Universal Robots URScript: vino 4binf.script

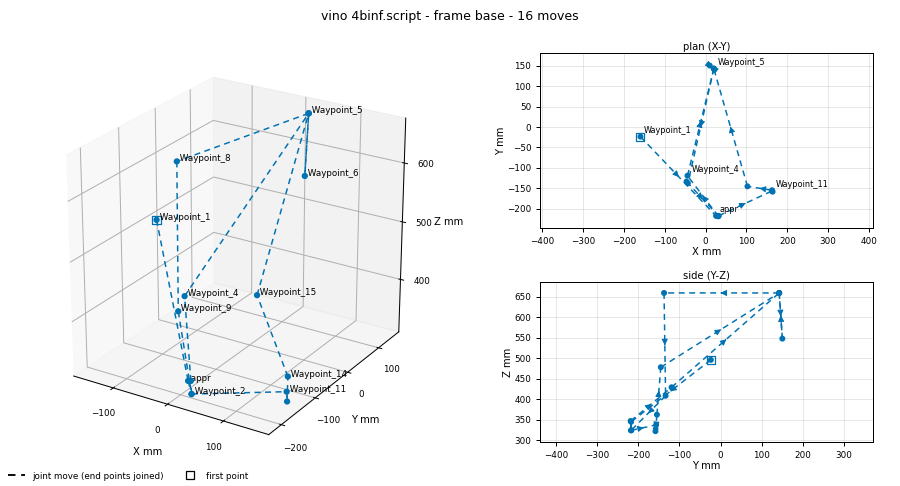
[picture p0: tool path of vino 4binf.script in frame base, 16 of 17 moves have a stored position in this frame; points joined in program order, loops and branches not executed]
def vino_4binf():
  set_gravity([0.0, 0.0, 9.82])
  set_safety_mode_transition_hardness(1)
  step_count_7828767f_f0a1_4da8_ad6d_1d539f3a6eb4 = 0.0
  thread Step_Counter_Thread_a07dad3b_d2d5_4c2a_9756_74ff32e0ed35():
    while (True):
      step_count_7828767f_f0a1_4da8_ad6d_1d539f3a6eb4 = step_count_7828767f_f0a1_4da8_ad6d_1d539f3a6eb4 + 1.0
      sync()
    end
  end
  run Step_Counter_Thread_a07dad3b_d2d5_4c2a_9756_74ff32e0ed35()
  set_tcp(p[0.0,0.0,0.155,0.0,0.0,0.0])
  set_payload(1.1, [0.0, 0.0, 0.06])
  set_standard_analog_input_domain(0, 1)
  set_standard_analog_input_domain(1, 1)
  set_tool_analog_input_domain(0, 1)
  set_tool_analog_input_domain(1, 1)
  set_analog_outputdomain(0, 0)
  set_analog_outputdomain(1, 0)
  set_input_actions_to_default()
  set_tool_voltage(24)
  global Plane_obliquo=p[0.09998422840375992,0.0999895685224925,0.14997740118490663,-0.1474295993751028,-0.061308860415087624,0.7833703634583852]
  global Plane_orizz=p[9.515322773469715E-6,0.2500097097193357,0.14997678393289224,-8.204102312405902E-5,-5.45201065398691E-5,1.2537983658861858E-5]
  global Plane_vert=p[2.5528049992290395E-5,0.45000115403946234,0.014993315552056186,1.5707062492170034,-1.3296462557657132E-4,1.823233379452444E-4]
  # begin: URCap Installation Node
  #   Source: OnRobot, 6.0.3, OnRobot A/S
  #   Type: OnRobot Setup
  sleep(1)
  if (False):
    global sg_Busy = 0
    global sg_Depth = 0
    global sg_Width = 0
  end
  ON_CONN_SHIFT_BOOL = 64
  ON_CONN_SHIFT_INT = 24
  ON_CONN_SHIFT_FLOAT = 24
  ON_CONN_REG_SUM_BOOL = 2
  ON_CONN_REG_SUM_INT = 4
  ON_CONN_REG_SUM_FLOAT = 3
  ON_TOOL_SHIFT_BOOL = 64
  ON_TOOL_SHIFT_INT = 25
  ON_TOOL_SHIFT_FLOAT = 24
  ON_TOOL_SHIFT_BOOL_ARR = [64, 66, 66]
  ON_TOOL_SHIFT_INT_ARR = [25, 28, 28]
  ON_TOOL_SHIFT_FLOAT_ARR = [24, 27, 27]
  ON_TOOL_REG_SUM_BOOL = 2
  ON_TOOL_REG_SUM_INT = 3
  ON_TOOL_REG_SUM_FLOAT = 3
  ON_REGISTERS_SPEEDL_FLOAT = 0
  ON_REG_USE_TOOL = False
  ON_DI_SINGLE = 0
  ON_DI_PRIMARY = 1
  ON_DI_SECONDARY = 2
  ON_DI_DUAL = 3
  on_robot_type = 3
  on_robot_cycle = 8.0
  on_conn_ip = "localhost"
  on_tool_ip = "localhost"
  on_device_socket_port = 51234
  on_conn_xmlrpc = rpc_factory("xmlrpc", "http://localhost:41414")
  on_tool_xmlrpc = rpc_factory("xmlrpc", "http://localhost:41414")
  on_RPC = rpc_factory("xmlrpc", "http://127.0.0.1:31416")
  ON_DEBUG_LOG = False
  on_isMetric = True
  on_toolConnector = True
  on_ioqc = True
  on_dual = False
  on_computebox = False
  on_devices = 1
  on_gripper = [False, False, False]
  on_custom_tcp_id = "none"
  on_custom_tcp_enabled = False
  speedlTime = 0.001
  on_ft = False
  sg_index = 0
  on_gripper[sg_index] = True
  #======    OnRobot Globals    ======#

  ON_MATH_PI=3.141593
  ON_ZEROPOSE=p[0.0,0.0,0.0,0.0,0.0,0.0]
  ON_ZEROFRAME=p[0.0,0.0,0.0,0.0,0.0,0.0]
  ON_ZERO3D=[0.0,0.0,0.0]
  ON_ZERO6D=[0.0,0.0,0.0,0.0,0.0,0.0]
  ON_ZERO8D=[0.0,0.0,0.0,0.0,0.0,0.0,0.0,0.0]
  ON_FALSE3D=[False,False,False]
  ON_FALSE6D=[False,False,False,False,False,False]
  ON_FALSE8D=[False,False,False,False,False,False,False,False]
  global on_return=0
  on_speedL=ON_ZERO6D
  on_speedBase=ON_ZERO6D
  on_speedVect=ON_ZERO6D
  on_speedExtra=ON_ZERO6D
  on_speedCB=ON_ZERO6D
  on_speedGecko=ON_ZERO6D
  on_RTDE_error=0
  on_RTDE_tool_error=0
  on_dataProcess_thrd=0
  ON_DEVICE_ID_MISSING=0
  ON_INIT_WATCHDOG_HZ=5
  ON_INIT_TIMEOUT=2000
  on_robot_TCP_offset=ON_ZEROFRAME
  on_tcp_offset_actual=ON_ZEROFRAME
  on_cog_actual=ON_ZEROFRAME
  on_mass_actual=0.0
  on_robot_mount=[0.0,0.0]

  #======    End of OnRobot Globals    ======#
  #======    OnRobot SG Globals    ======#

  SG_DEVICE_ID=80
  sg_Width_arr=[0,0,0]
  sg_Depth_arr=[0,0,0]
  sg_DepthRel_arr=[0,0,0]
  sg_device_id_arr=[0,0,0]
  sg_product_code_arr=[0,0,0]
  sg_Status_arr=[0,0,0]
  sg_Busy_arr=[False,False,False]
  sg_Initialized_arr=[False,False,False]
  sg_Grip_command_arr=[False,False,False]
  sg_tool_id_arr=[0,0,0]

  sg_Width=0
  sg_Depth=0
  sg_Busy=False
  def get_sg_Width():
  return sg_Width
  end
  def get_sg_Depth():
  return sg_Depth
  end
  def get_sg_Busy():
  return sg_Busy
  end


  #======    End of OnRobot SG Globals    ======#
  #======    OnRobot Interface Messages    ======#

  on_devices_primary_log="OnRobot Devices"
  on_devices_secondary_log="OnRobot Secondary Device"
  on_program_halted="<br>Program halted."
  on_device_error_title="OnRobot - Device error"
  on_install_error="OnRobot Setup is not correct.<br>Check the status in the OnRobot Setup page in the Installation Tab.<br>Program halted."
  on_device_missing="No device connected.<br>Program halted."
  cb_device_missing="No OnRobot Compute Box connected.<br>Program halted."
  ft_device_missing="No OnRobot FT sensor or license detected.<br>Program halted."
  hex_device_missing="No HEX sensor connected.<br>Program halted."
  rg2ft_device_missing="No RG2-FT gripper connected.<br>Program halted."
  rg_device_missing="No RG gripper connected.<br>Program halted."
  vg_device_missing="No VG gripper connected.<br>Program halted."
  gg_device_missing="No Gecko Gripper connected.<br>Program halted."
  sg_device_missing="No Soft Gripper connected.<br>Program halted."
  tfg_device_missing="No 3FG gripper connected.<br>Program halted."
  sdr_device_missing="No OnRobot Sander connected.<br>Program halted."
  twofg_device_missing="No 2FG gripper connected.<br>Program halted."
  vgp_device_missing="No VGP gripper connected.<br>Program halted."
  mg_device_missing="No Magnetic Gripper connected.<br>Program halted."
  fgp_device_missing="No 2FGP20 Gripper connected.<br>Program halted."
  eyes_device_missing="No OnRobot Eyes connected.<br>Program halted."
  on_xmlrpc_start_ip="Connecting to OnRobot XML-RPC Server:"
  on_java_comm_error_textmsg_title="OnRobot - Communication error:"
  on_java_comm_controlsocket_open_error="Socket 'javaSocket' opening was unsuccessful."
  on_java_comm_error_title="OnRobot - Communication error"
  on_java_comm_socket_open_error="Establishing connection with the URCap was timed out.<br>Check the status in the OnRobot Setup page in the Installation Tab.<br>Program halted."
  on_rtde_feed_error_textmsg_title="OnRobot - RTDE error:"
  on_rtde_feed_error="RTDE feed error. OnRobot device count mismatch.<br>Program halted."
  on_rtde_feed_tool_error="Tool RTDE feed error. OnRobot device count mismatch.<br>Program halted."
  on_rtde_feed_open_error_textmsg="Socket 'rtdeFeed' opening was unsuccessful."
  on_rtde_feed_error_title="OnRobot - RTDE error"
  on_rtde_feed_count_error="Invalid RTDE offset setup detected. Please check RTDE Offsets at the OnRobot Setup page in the Installation Tab.<br>Program halted."
  on_rtde_feed_open_error="Establishing connection with the devices was timed out.<br>Ensure that the OnRobot devices are operational, and check the status in the OnRobot Setup page in the Installation Tab."

  #======    End of OnRobot Interface Messages    ======#
  #======    OnRobot Interface    ======#

  on_portopened_javaSocket=False
  on_rtde_feed_opened=False
  on_dataProcess_running=False
  def on_missing():
  popup(on_device_missing,title=on_device_error_title,error=True,blocking=False)
  halt
  end
  def cb_missing():
  popup(cb_device_missing,title=on_device_error_title,error=True,blocking=False)
  halt
  end
  def ft_missing():
  popup(ft_device_missing,title=on_device_error_title,error=True,blocking=False)
  halt
  end
  def hex_missing():
  popup(hex_device_missing,title=on_device_error_title,error=True,blocking=False)
  halt
  end
  def rg2ft_missing():
  popup(rg2ft_device_missing,title=on_device_error_title,error=True,blocking=False)
  halt
  end
  def rg_missing():
  popup(rg_device_missing,title=on_device_error_title,error=True,blocking=False)
  halt
  end
  def vg_missing():
  popup(vg_device_missing,title=on_device_error_title,error=True,blocking=False)
  halt
  end
  def gg_missing():
  popup(gg_device_missing,title=on_device_error_title,error=True,blocking=False)
  halt
  end
  def sg_missing():
  popup(sg_device_missing,title=on_device_error_title,error=True,blocking=False)
  halt
  end
  def tfg_missing():
  popup(tfg_device_missing,title=on_device_error_title,error=True,blocking=False)
  halt
  end
  def sdr_missing():
  popup(sdr_device_missing,title=on_device_error_title,error=True,blocking=False)
  halt
  end
  def twofg_missing():
  popup(twofg_device_missing,title=on_device_error_title,error=True,blocking=False)
  halt
  end
  def vgp_missing():
  popup(vgp_device_missing,title=on_device_error_title,error=True,blocking=False)
  halt
  end
  def mg_missing():
  popup(mg_device_missing,title=on_device_error_title,error=True,blocking=False)
  halt
  end
  def fgp_missing():
  popup(fgp_device_missing,title=on_device_error_title,error=True,blocking=False)
  halt
  end
  def eyes_missing():
  popup(eyes_device_missing,title=on_device_error_title,error=True,blocking=False)
  halt
  end
  def on_portclose_javaSocket():
  socket_close("javaSocket")
  on_portopened_javaSocket=False
  end
  def on_portopen_javaSocket():
  on_portclose_javaSocket()
  on_portopened_javaSocket=socket_open("127.0.0.1",44005,"javaSocket")
  if not on_portopened_javaSocket:
  textmsg(on_java_comm_error_textmsg_title,on_java_comm_controlsocket_open_error)
  popup(on_java_comm_socket_open_error,title=on_java_comm_error_title,error=True,blocking=False)
  halt
  end
  end
  on_conn_rtde_feed_name="rtdeFeedConn"
  on_tool_rtde_feed_name="rtdeFeedTool"
  def on_rtde_feed_close(rtdeFeedName):
  socket_close(rtdeFeedName)
  on_rtde_feed_opened=False
  end
  def on_rtde_feed_open(deviceIP,rtdeFeedName,regStart,regSum,regSpeedl):
  on_rtde_feed_close(rtdeFeedName)
  if((regStart[0]+regSum[0])>128)or((regStart[1]+regSum[1])>48)or((regStart[2]+regSum[2])>48):
  popup(on_rtde_feed_count_error,title=on_rtde_feed_error_title,error=True,blocking=False)
  textmsg(str_cat("RegStart: ",regStart),str_cat("  -  RegSum: ",regSum))
  halt
  end
  on_rtde_feed_opened=socket_open(deviceIP,on_device_socket_port,rtdeFeedName)
  if not on_rtde_feed_opened:
  on_rtde_feed_opened=socket_open(deviceIP,on_device_socket_port,rtdeFeedName)
  end
  if not on_rtde_feed_opened:
  textmsg(on_rtde_feed_error_textmsg_title,on_rtde_feed_open_error_textmsg)
  popup(on_rtde_feed_open_error,title=on_rtde_feed_error_title,error=True,blocking=False)
  halt
  end
  socket_send_int(regStart[0],rtdeFeedName)
  socket_send_int(regSum[0],rtdeFeedName)
  socket_send_int(regStart[1],rtdeFeedName)
  socket_send_int(regSum[1],rtdeFeedName)
  socket_send_int(regStart[2],rtdeFeedName)
  socket_send_int(regSum[2],rtdeFeedName)
  socket_send_int(regSpeedl,rtdeFeedName)
  socket_send_int(on_devices,rtdeFeedName)
  end
  def on_dataRead():
  enter_critical
  on_RTDE_error=read_input_integer_register(ON_CONN_SHIFT_INT)
  if(ON_REG_USE_TOOL):
  on_RTDE_tool_error=read_input_integer_register(ON_TOOL_SHIFT_INT_ARR[0])
  end
  exit_critical
  end
  def on_set_rtde_watchdog(updateHz=ON_INIT_WATCHDOG_HZ):
  local effect="stop"
  if(updateHz<1):
  effect="ignore"
  end
  watchdog_conn_reg_str=str_cat("input_int_register_",ON_CONN_SHIFT_INT)
  rtde_set_watchdog(watchdog_conn_reg_str,updateHz,effect)
  if(ON_REG_USE_TOOL):
  watchdog_tool_reg_str=str_cat("input_int_register_",ON_TOOL_SHIFT_INT_ARR[0])
  rtde_set_watchdog(watchdog_tool_reg_str,updateHz,effect)
  end
  if ON_DEBUG_LOG:
  local update_str=str_cat(" "+effect+" watchdog set to [Hz]: ",updateHz)
  textmsg(watchdog_conn_reg_str,update_str)
  if(ON_REG_USE_TOOL):
  local update_str=str_cat(" "+effect+" watchdog set to [Hz]: ",updateHz)
  textmsg(watchdog_tool_reg_str,update_str)
  end
  end
  end
  def on_speedCB_get():
  return[on_speedCB[0],on_speedCB[1],on_speedCB[2],on_speedCB[3],on_speedCB[4],on_speedCB[5]]
  end
  def on_speedGecko_get():
  local speedExtra=ON_ZERO6D
  if on_speedl_for_gecko:
  speedExtra=[on_speedGecko[0],on_speedGecko[1],on_speedGecko[2],on_speedGecko[3],on_speedGecko[4],on_speedGecko[5]]
  end
  return speedExtra
  end
  def on_speedGecko_set(speedGecko):
  on_speedGecko=[speedGecko[0],speedGecko[1],speedGecko[2],speedGecko[3],speedGecko[4],speedGecko[5]]
  end
  thread on_dataProcess_thread():
  if ON_DEBUG_LOG:
  textmsg("Starting on_dataRead thread")
  end
  local error=False
  on_dataProcess_running=True
  sync()
  while on_dataProcess_running:
  sync()
  on_dataRead()
  error=on_error((on_RTDE_error<0),on_rtde_feed_error,on_rtde_feed_error_title,error)
  error=on_error((ON_REG_USE_TOOL and(on_RTDE_tool_error<0)),on_rtde_feed_tool_error,on_rtde_feed_error_title,error)
  on_dataProcess_running=not error
  end
  if error:
  halt
  end
  if ON_DEBUG_LOG:
  textmsg("Stopping on_dataRead thread")
  end
  end
  thread on_set_watchdog_thread():
  sleep(2)
  on_set_rtde_watchdog(updateHz=ON_INIT_WATCHDOG_HZ)
  sleep(1/ON_INIT_WATCHDOG_HZ)
  on_dataProcess_running=False
  kill on_dataProcess_thrd
  end

  #======    End of OnRobot Interface    ======#
  #======    OnRobot QC Setup Tool Connector    ======#

  def tc_setup_tool():
  if ON_DEBUG_LOG:
  textmsg("QC Setup Tool Connector start...")
  end
  set_tool_voltage(24)

  if ON_DEBUG_LOG:
  textmsg("QC Setup Tool Connector end.")
  end
  end

  #======    End of OnRobot QC Setup Tool Connector    ======#
  #======    OnRobot SG Interface    ======#

  sg_dataRead_running=False
  def sg_dataRead_RTDE(tool_index):
  local reg_offset_bool=ON_TOOL_SHIFT_BOOL_ARR[tool_index]
  local reg_offset_int=ON_TOOL_SHIFT_INT_ARR[tool_index]
  local reg_offset_float=ON_TOOL_SHIFT_FLOAT_ARR[tool_index]
  enter_critical
  floatRegDummy=read_input_float_register(reg_offset_float+0)
  sg_Width_arr[tool_index]=floatRegDummy
  floatRegDummy=read_input_float_register(reg_offset_float+1)
  sg_Depth_arr[tool_index]=floatRegDummy
  floatRegDummy=read_input_float_register(reg_offset_float+2)
  sg_DepthRel_arr[tool_index]=floatRegDummy
  intRegDummy=read_input_integer_register(reg_offset_int+0)
  sg_device_id_arr[tool_index]=intRegDummy
  intRegDummy=read_input_integer_register(reg_offset_int+1)
  sg_product_code_arr[tool_index]=intRegDummy
  intRegDummy=read_input_integer_register(reg_offset_int+2)
  sg_Status_arr[tool_index]=intRegDummy
  boolRegDummy=read_input_boolean_register(reg_offset_bool+0)
  sg_Busy_arr[tool_index]=boolRegDummy
  boolRegDummy=read_input_boolean_register(reg_offset_bool+1)
  sg_Initialized_arr[tool_index]=boolRegDummy
  exit_critical
  end
  thread sg_dataRead_thread():
  if ON_DEBUG_LOG:
  textmsg("Starting sg_dataRead thread")
  end
  while sg_dataRead_running:
  sync()
  if(sg_index==ON_DI_DUAL):
  sg_dataRead_RTDE(ON_DI_PRIMARY)
  sg_dataRead_RTDE(ON_DI_SECONDARY)
  else:
  sg_dataRead_RTDE(sg_index)
  end
  end
  if ON_DEBUG_LOG:
  textmsg("Stopping sg_dataRead thread")
  end
  end

  #======    End of OnRobot SG Interface    ======#
  #======    OnRobot TCP Messages    ======#

  on_tcp_log_msg_default="OnRobot: Robot TCP Offset set to:"
  on_tcp_log_msg_primary="OnRobot: Robot TCP Offset set to Primary:"
  on_tcp_log_msg_secondary="OnRobot: Robot TCP Offset set to Secondary:"

  #======    End of OnRobot TCP Messages    ======#
  #======    OnRobot TCP    ======#

  on_tcp_offset_actual=ON_ZEROFRAME
  on_tcp_offset_primary=ON_ZEROFRAME
  on_tcp_static_primary=ON_ZEROFRAME
  on_tcp_dynamic_primary=ON_ZEROFRAME
  on_tcp_adapters=ON_ZEROFRAME
  on_tcp_qc_primary=ON_ZEROFRAME
  on_tcp_base_primary=ON_ZEROFRAME
  on_tcp_gripper_static_primary=ON_ZEROFRAME
  on_tcp_workpiece_primary=ON_ZEROFRAME
  on_tcp_gripper_dynamic_primary=ON_ZEROFRAME
  on_tcp_gripper_primary=ON_ZEROFRAME
  on_tcp_offset_secondary=ON_ZEROFRAME
  on_tcp_static_secondary=ON_ZEROFRAME
  on_tcp_dynamic_secondary=ON_ZEROFRAME
  on_tcp_qc_secondary=ON_ZEROFRAME
  on_tcp_base_secondary=ON_ZEROFRAME
  on_tcp_gripper_static_secondary=ON_ZEROFRAME
  on_tcp_workpiece_secondary=ON_ZEROFRAME
  on_tcp_gripper_dynamic_secondary=ON_ZEROFRAME
  on_tcp_gripper_secondary=ON_ZEROFRAME
  on_tcp_custom_preset_assigned=False
  on_tcp_custom_preset=ON_ZEROFRAME
  def on_tcp_init_adapters():
  if ON_DEBUG_LOG:
  textmsg("TCP Init Adapters start..")
  end
  enter_critical
  on_tcp_adapters=ON_ZEROFRAME
  local adapterCount=length(on_tcp_adapters_array)
  local i=0
  while(i<adapterCount):
  on_tcp_adapters=pose_trans(on_tcp_adapters,on_tcp_adapters_array[i])
  i=i+1
  end
  exit_critical
  if ON_DEBUG_LOG:
  textmsg("TCP Init Adapters end.")
  end
  end
  def on_tcp_update_primary():
  if ON_DEBUG_LOG:
  textmsg("TCP Update Primary start..")
  end
  on_tcp_gripper_dynamic_primary=p[0.0, 0.0, 0.0, 0.0, 0.0, 0.0]
  enter_critical
  on_tcp_dynamic_primary=pose_trans(on_tcp_static_primary,on_tcp_gripper_dynamic_primary)
  on_tcp_offset_primary=pose_trans(on_tcp_dynamic_primary,on_tcp_workpiece_primary)
  exit_critical
  if ON_DEBUG_LOG:
  textmsg("TCP Update Primary end.")
  end
  end
  def on_tcp_init_primary():
  if ON_DEBUG_LOG:
  textmsg("TCP Init Primary start..")
  end
  enter_critical
  on_tcp_base_primary=pose_trans(on_tcp_adapters,on_tcp_qc_primary)
  on_tcp_static_primary=pose_trans(on_tcp_base_primary,on_tcp_gripper_static_primary)
  exit_critical
  on_tcp_update_primary()
  if ON_DEBUG_LOG:
  textmsg("TCP Init Primary end.")
  end
  end
  def on_tcp_offset_set(TCP_offset):
  if ON_DEBUG_LOG:
  textmsg("TCP Offset set started!")
  end
  on_tcp_offset_send(TCP_offset)
  if(on_follow_tcp):
  set_tcp(TCP_offset)
  end
  on_robot_TCP_offset=TCP_offset
  if ON_DEBUG_LOG:
  textmsg("TCP Offset set to: ",on_robot_TCP_offset)
  end
  end
  def on_tcp_offset_forced_set_actual(isPrimary=True):
  if(not on_follow_tcp):

  local tcp_log_msg=on_tcp_log_msg_default

  textmsg(tcp_log_msg,on_tcp_offset_actual)
  set_tcp(on_tcp_offset_actual)
  end
  end
  def on_tcp_update(isPrimary=True):
  on_tcp_update_primary()

  on_tcp_set_actual_to(isPrimary)
  end
  def on_tcp_set_actual_to(isPrimary=True):

  on_tcp_offset_actual=on_tcp_offset_primary
  if(on_follow_tcp):
  textmsg(on_tcp_log_msg_default,on_tcp_offset_actual)
  end

  on_tcp_active_is_primary=isPrimary
  on_tcp_offset_set(on_tcp_offset_actual)
  end
  def on_tcp_update_workpiece_primary(workpiece_offset):
  if ON_DEBUG_LOG:
  textmsg("TCP Update Tool Primary start..")
  end
  on_tcp_workpiece_primary=workpiece_offset
  on_tcp_update_primary()
  if ON_DEBUG_LOG:
  textmsg("TCP Update Tool Primary end.")
  end
  end
  def on_tcp_workpiece_rpy_get(xyz=[0.0,0.0,0.0],rpy=[0.0,0.0,0.0]):
  local rotvec=rpy2rotvec(rpy)
  local workpiece_offset=p[xyz[0],xyz[1],xyz[2],rotvec[0],rotvec[1],rotvec[2]]
  return workpiece_offset
  end

  def on_tcp_update_workpiece(workpiece_offset,tool_index=0):
  if ON_DEBUG_LOG:
  textmsg("TCP Update Tool start..")
  end
  if(tool_index!=ON_DI_SECONDARY):
  on_tcp_update_workpiece_primary(workpiece_offset)
  local isPrimary=True

  end
  on_tcp_set_actual_to(isPrimary)
  if ON_DEBUG_LOG:
  textmsg("TCP Update Tool end.")
  end
  end
  def on_get_tcp_for(tool_index):
  if tool_index==ON_DI_SECONDARY:
  local actual_tcp=on_tcp_static_secondary
  else:
  local actual_tcp=on_tcp_static_primary
  end
  return actual_tcp
  end
  def on_tcp_custom_unused():
  return ON_ZEROFRAME
  end
  def on_tcp_update_custom():
  if ON_DEBUG_LOG:
  textmsg("TCP Update Custom start..")
  end
  if(on_custom_tcp_enabled):
  on_tcp_custom_unused()
  on_tcp_custom_unused()
  on_tcp_custom_unused()
  on_tcp_custom_unused()

  end
  if ON_DEBUG_LOG:
  textmsg("TCP Update Custom end.")
  end
  end

  #======    End of OnRobot TCP    ======#
  #======    OnRobot Payload Messages    ======#

  on_mass_log_msg="OnRobot: Robot Payload Mass set to:"
  on_cog_log_msg="OnRobot: Robot Payload Center of Gravity set to:"

  #======    End of OnRobot Payload Messages    ======#
  #======    OnRobot Payload    ======#

  on_cog_actual=ON_ZEROFRAME
  on_mass_actual=0.0
  on_cog_primary=ON_ZEROFRAME
  on_cog_L1L2_primary=ON_ZEROFRAME
  on_mass_primary=0.0
  on_mass_L1L2_primary=0.0
  on_cog_adapters=ON_ZEROFRAME
  on_cog_qc_primary=ON_ZEROFRAME
  on_cog_base_primary=ON_ZEROFRAME
  on_cog_gripper_primary=ON_ZEROFRAME
  on_cog_workpiece_primary=ON_ZEROFRAME
  on_mass_adapters=0.0
  on_mass_qc_primary=0.0
  on_mass_base_primary=0.0
  on_mass_gripper_primary=0.0
  on_mass_workpiece_primary=0.0
  on_cog_secondary=ON_ZEROFRAME
  on_mass_secondary=0.0
  on_cog_gripper_secondary=ON_ZEROFRAME
  on_mass_gripper_secondary=0.0
  on_cog_workpiece_secondary=ON_ZEROFRAME
  on_mass_workpiece_secondary=0.0
  ON_LB2KG001=0.45359237/100
  def on_payload_init_adapters():
  if ON_DEBUG_LOG:
  textmsg("TCP Init Adapters start..")
  end
  enter_critical
  on_cog_adapters=ON_ZEROFRAME
  on_mass_adapters=0.0
  local massLAL0Ratio=0
  local adapterAbsCOG=ON_ZEROFRAME
  local tcp_adapter_offset=ON_ZEROFRAME
  local adapterCount=length(on_tcp_adapters_array)
  local i=0
  while(i<adapterCount):
  on_mass_adapters=on_mass_adapters+on_mass_adapters_array[i]
  if(on_mass_adapters<=0):
  massLAL0Ratio=0
  else:
  massLAL0Ratio=on_mass_adapters_array[i]/on_mass_adapters
  end
  adapterAbsCOG=pose_trans(tcp_adapter_offset,on_tcp_adapters_array[i])
  adapterAbsCOG=p[adapterAbsCOG[0],adapterAbsCOG[1],adapterAbsCOG[2],0.0,0.0,0.0]
  on_cog_adapters=interpolate_pose(on_cog_adapters,adapterAbsCOG,massLAL0Ratio)
  on_cog_adapters=p[on_cog_adapters[0],on_cog_adapters[1],on_cog_adapters[2],0.0,0.0,0.0]
  tcp_adapter_offset=pose_trans(tcp_adapter_offset,on_tcp_adapters_array[i])
  i=i+1
  sync()
  end
  exit_critical
  if ON_DEBUG_LOG:
  textmsg("TCP Init Adapters end.")
  end
  end
  def on_payload_update_primary():
  if ON_DEBUG_LOG:
  textmsg("Payload Update Primary start..")
  end
  enter_critical
  on_mass_primary=on_mass_L1L2_primary+on_mass_workpiece_primary
  local massL1L2L3Ratio=on_mass_workpiece_primary/on_mass_primary
  local workpieceAbsCOG=pose_trans(on_tcp_dynamic_primary,on_cog_workpiece_primary)
  workpieceAbsCOG=p[workpieceAbsCOG[0],workpieceAbsCOG[1],workpieceAbsCOG[2],0.0,0.0,0.0]
  on_cog_primary=interpolate_pose(on_cog_L1L2_primary,workpieceAbsCOG,massL1L2L3Ratio)
  on_cog_primary=p[on_cog_primary[0],on_cog_primary[1],on_cog_primary[2],0.0,0.0,0.0]
  exit_critical
  if ON_DEBUG_LOG:
  textmsg("Payload Update Primary end.")
  end
  end
  def on_payload_init_primary():
  if ON_DEBUG_LOG:
  textmsg("Payload Init Primary start..")
  end
  enter_critical
  on_mass_base_primary=on_mass_adapters+on_mass_qc_primary
  local massL0L1Ratio=on_mass_qc_primary/on_mass_base_primary
  on_mass_L1L2_primary=on_mass_base_primary+on_mass_gripper_primary
  local massL1L2Ratio=on_mass_gripper_primary/on_mass_L1L2_primary
  local qcAbsCOG=pose_trans(on_tcp_adapters,on_cog_qc_primary)
  qcAbsCOG=p[qcAbsCOG[0],qcAbsCOG[1],qcAbsCOG[2],0.0,0.0,0.0]
  on_cog_base_primary=interpolate_pose(on_cog_adapters,qcAbsCOG,massL0L1Ratio)
  on_cog_base_primary=p[on_cog_base_primary[0],on_cog_base_primary[1],on_cog_base_primary[2],0.0,0.0,0.0]
  local gripperAbsCOG=pose_trans(on_tcp_base_primary,on_cog_gripper_primary)
  gripperAbsCOG=p[gripperAbsCOG[0],gripperAbsCOG[1],gripperAbsCOG[2],0.0,0.0,0.0]
  on_cog_L1L2_primary=interpolate_pose(on_cog_base_primary,gripperAbsCOG,massL1L2Ratio)
  on_cog_L1L2_primary=p[on_cog_L1L2_primary[0],on_cog_L1L2_primary[1],on_cog_L1L2_primary[2],0.0,0.0,0.0]
  exit_critical
  on_payload_update_primary()
  if ON_DEBUG_LOG:
  textmsg("Payload Init Primary end.")
  end
  end
  def on_payload_update():
  on_payload_update_primary()

  on_mass_actual =on_mass_primary
  on_cog_actual=on_cog_primary

  on_payload_set_actual()
  end
  def on_payload_set_actual():

  on_mass_actual =on_mass_primary
  on_cog_actual=on_cog_primary

  local CoG=[on_cog_actual[0],on_cog_actual[1],on_cog_actual[2]]
  on_payload_set(on_mass_actual,CoG)
  end
  def on_payload_update_workpiece_primary(workpiece_mass=0,workpiece_cog=[0.0,0.0,0.0]):
  if ON_DEBUG_LOG:
  textmsg("Payload Update Workpiece Primary start..")
  end
  on_cog_workpiece_primary=p[workpiece_cog[0],workpiece_cog[1],workpiece_cog[2],0.0,0.0,0.0]
  on_mass_workpiece_primary=workpiece_mass
  on_payload_update_primary()
  if ON_DEBUG_LOG:
  textmsg("Payload Update Workpiece Primary end.")
  end
  end
  def on_payload_set(mass,CoG):
  if ON_DEBUG_LOG:
  textmsg("Payload set started!")
  end
  local center_of_gravity=[CoG[0],CoG[1],CoG[2]]
  on_payload_send(center_of_gravity,mass)
  if(on_isMetric):
  local roundedMass=floor(mass*100+0.5)/100
  else:
  local roundedMass=floor(mass/ON_LB2KG001+0.5)*ON_LB2KG001
  end
  set_payload(roundedMass,center_of_gravity)
  on_mass_actual=roundedMass
  on_cog_actual=p[CoG[0],CoG[1],CoG[2],0.0,0.0,0.0]
  if ON_DEBUG_LOG:
  textmsg("Payload mass, CoG set to: ",str_cat(str_cat(mass,", "),CoG))
  end
  end

  def on_payload_update_secondary():
  end
  def on_payload_init_secondary():
  end

  def on_payload_update_workpiece(workpiece_mass,workpiece_cog=[0.0,0.0,0.0],tool_index=0):
  if ON_DEBUG_LOG:
  textmsg("Payload Update Workpiece start..")
  end
  if(tool_index!=ON_DI_SECONDARY):
  on_cog_workpiece_primary=p[workpiece_cog[0],workpiece_cog[1],workpiece_cog[2],0.0,0.0,0.0]
  on_mass_workpiece_primary=workpiece_mass
  else:
  on_cog_workpiece_secondary=p[workpiece_cog[0],workpiece_cog[1],workpiece_cog[2],0.0,0.0,0.0]
  on_mass_workpiece_secondary=workpiece_mass
  end
  on_payload_update()
  if ON_DEBUG_LOG:
  textmsg("Payload Update Workpiece end.")
  end
  end
  def on_payload_get_cog2tcp_workpiece(tool_index=0):
  if(tool_index!=ON_DI_SECONDARY):
  local cog_tool=[on_tcp_workpiece_primary[0],on_tcp_workpiece_primary[1],on_tcp_workpiece_primary[2]]
  else:
  local cog_tool=[on_tcp_workpiece_secondary[0],on_tcp_workpiece_secondary[1],on_tcp_workpiece_secondary[2]]
  end
  return cog_tool
  end

  #======    End of OnRobot Payload    ======#
  #======    OnRobot QC TCP    ======#

  onrobotmini=0

  def on_tcp_offset_send(TCP_offset):
  on_robot_TCP_offset=TCP_offset
  end
  def on_payload_send(CoG,mass):
  on_robot_payload_cog=CoG
  on_robot_payload_mass=mass
  end


  #======    End of OnRobot QC TCP    ======#
  #======    OnRobot SG TCP    ======#

  def sg_tcp_dynamic_get(tool_index=0):
  local gripperDepth=sg_Depth_arr[tool_index]
  local z_offset=-gripperDepth/1000.0
  return p[0.0,0.0,z_offset,0.0,0.0,0.0]
  end
  def sg_tcp_static_silicone_get(tool_index=0):
  local baseUnitStatic=89
  local gripperStaticDepth=on_tool_xmlrpc.sg_get_depth_static_silicone(tool_index)+baseUnitStatic
  local z_offset=gripperStaticDepth/1000.0
  return p[0.0,0.0,z_offset,0.0,0.0,0.0]
  end
  def sg_payload_set(mass,tool_index=0):
  if ON_DEBUG_LOG:
  textmsg("SG Payload mass command starting..")
  end
  if(tool_index==ON_DI_SECONDARY):
  local cogTool=[on_cog_workpiece_secondary[0],on_cog_workpiece_secondary[1],on_cog_workpiece_secondary[2]]
  else:
  local cogTool=[on_cog_workpiece_primary[0],on_cog_workpiece_primary[1],on_cog_workpiece_primary[2]]
  end
  if(sg_Grip_command_arr[tool_index]):
  local mass2set=mass
  else:
  local mass2set=0.0
  end
  on_payload_update_workpiece(mass2set,cogTool,tool_index)
  if ON_DEBUG_LOG:
  textmsg("SG Payload mass command ended.")
  end
  end

  #======    End of OnRobot SG TCP    ======#
  #======    OnRobot  Speedl    ======#

  on_speedl_thread_handler=0
  on_speedl_is_enabled=False
  on_speedl_is_running=False
  on_speedl_acc=0.0
  ft_speedl_hg_caranteen_reached=False
  ft_speedl_hg_caranteen_safemode=False
  on_speedl_for_ftcontrol=False
  on_speedl_for_move=False
  on_speedl_for_handguide=False
  on_speedl_for_insertpart=False
  on_speedl_for_depthcompensation=False
  on_speedl_for_center=False
  on_speedl_for_gecko=False
  on_speedl_acc=10000.0
  on_speedl_acc_to_zero=3.0
  ON_SPEEDL_FTCONTROL=1
  ON_SPEEDL_HANDGUIDE=2
  ON_SPEEDL_TRAJECTORY=3
  ON_SPEEDL_MOVE=ON_SPEEDL_TRAJECTORY
  ON_SPEEDL_INSERTPART=4
  ON_SPEEDL_DEPTHCOMP=5
  ON_SPEEDL_CENTER=6
  ON_SPEEDL_GECKO=7
  def on_wait_ms(time_ms):
  local sync_time=ceil(norm(time_ms/8.0))
  while(sync_time>0):
  sync_time=sync_time-1
  sync()
  end
  end
  def on_error(status_flag,message,title,stop_var=False):
  if(status_flag):
  popup(message,title=title,error=True,blocking=False)
  stop_var=True
  end
  return stop_var
  end
  def on_warning(status_flag,message,title,isPopupNeeded=False,is_shown=False):
  if(status_flag):
  if(not is_shown):
  if(isPopupNeeded):
  popup(message,title=title,warning=True,blocking=False)
  else:
  textmsg(title+": ",message)
  end
  is_shown=True
  end
  else:
  is_shown=False
  end
  return is_shown
  end
  def on_speedl_add_extra(speedBase,speedExtra):
  speedSum=ON_ZERO6D
  speedBaseP=p[speedBase[0],speedBase[1],speedBase[2],speedBase[3],speedBase[4],speedBase[5]]
  speedExtraP=p[speedExtra[0],speedExtra[1],speedExtra[2],speedExtra[3],speedExtra[4],speedExtra[5]]
  speedSumP=pose_add(speedExtraP,speedBaseP)
  speedSum=[speedSumP[0],speedSumP[1],speedSumP[2],speedSumP[3],speedSumP[4],speedSumP[5]]
  return speedSum
  end

  thread on_speedl_thread():
  if ON_DEBUG_LOG:
  textmsg("Speedl thread started..")
  end
  enter_critical
  on_speedl_is_running=True
  on_speedl_is_enabled=True
  exit_critical
  on_speedL=ON_ZERO6D
  on_speedL_last=ON_ZERO6D

  while on_speedl_is_running:
  on_speedBase=on_speedCB_get()
  on_speedL=on_speedBase


  if on_speedl_is_enabled:
  if(on_speedL==ON_ZERO6D):
  on_speedL=[on_speedL_last[0]/100,on_speedL_last[1]/100,on_speedL_last[2]/100,on_speedL_last[3]/100,on_speedL_last[4]/100,on_speedL_last[5]/100]
  end
  speedl(on_speedL,a=on_speedl_acc,t=speedlTime)
  else:
  speedl(ON_ZERO6D,a=on_speedl_acc_to_zero,t=speedlTime)
  end
  on_speedL_last=on_speedL
  end

  on_speedL=ON_ZERO6D
  if ON_DEBUG_LOG:
  textmsg("Speedl thread ended.")
  end
  end
  def on_speedl_integer_get():
  local speedl_integer=binary_list_to_integer([on_speedl_for_ftcontrol,on_speedl_for_handguide,on_speedl_for_move,on_speedl_for_insertpart,on_speedl_for_depthcompensation,on_speedl_for_center,on_speedl_for_gecko])
  return speedl_integer
  end
  def on_speedl_start_for(speedl_id):
  if(speedl_id==ON_SPEEDL_FTCONTROL):
  on_speedl_for_ftcontrol=True
  elif(speedl_id==ON_SPEEDL_HANDGUIDE):
  on_speedl_for_handguide=True
  elif(speedl_id==ON_SPEEDL_TRAJECTORY):
  on_speedl_for_move=True
  elif(speedl_id==ON_SPEEDL_INSERTPART):
  on_speedl_for_insertpart=True
  elif(speedl_id==ON_SPEEDL_DEPTHCOMP):
  on_speedl_for_depthcompensation=True
  elif(speedl_id==ON_SPEEDL_CENTER):
  on_speedl_for_center=True
  elif(speedl_id==ON_SPEEDL_GECKO):
  on_speedl_for_gecko=True
  else:
  textmsg("Unknown Start speedl ID received: ",speedl_id)
  end
  local speedl_integer=on_speedl_integer_get()
  if not(speedl_integer==0):
  if not on_speedl_is_running:
  on_speedl_thread_handler=run on_speedl_thread()
  end
  end
  return on_speedl_is_running
  end
  def on_speedl_stop_for(speedl_id,brake=10,brakeRot=10):
  if(speedl_id==ON_SPEEDL_FTCONTROL):
  on_speedl_for_ftcontrol=False
  elif(speedl_id==ON_SPEEDL_HANDGUIDE):
  on_speedl_for_handguide=False
  elif(speedl_id==ON_SPEEDL_TRAJECTORY):
  on_speedl_for_move=False
  elif(speedl_id==ON_SPEEDL_INSERTPART):
  on_speedl_for_insertpart=False
  elif(speedl_id==ON_SPEEDL_DEPTHCOMP):
  on_speedl_for_depthcompensation=False
  elif(speedl_id==ON_SPEEDL_CENTER):
  on_speedl_for_center=False
  elif(speedl_id==ON_SPEEDL_GECKO):
  on_speedl_for_gecko=False
  on_speedGecko_set(ON_ZERO6D)
  else:
  textmsg("Unknown Stop speedl ID received: ",speedl_id)
  end
  local speedl_integer=on_speedl_integer_get()
  if(speedl_integer==0):
  if(on_speedl_is_running):
  kill on_speedl_thread_handler
  enter_critical
  on_speedl_is_running=False
  exit_critical

  end
  if ON_DEBUG_LOG:
  textmsg("Speedl thread stopped")
  end
  stopl(brake,brakeRot)
  end
  return on_speedl_is_running
  end
  def on_speedl_pause():
  on_speedl_is_enabled=False
  return on_speedl_integer_get()
  end
  def on_speedl_resume():
  on_speedl_is_enabled=True
  return on_speedl_integer_get()
  end

  #======    End of OnRobot  Speedl    ======#
  #======    OnRobot SG Engine Messages Messages    ======#

  sg_title="OnRobot - Soft Gripper"
  sg_error_title="OnRobot - Soft Gripper error"
  sg_status_error_title="OnRobot - SG Status error"
  sg_status_error_missing="Communication problem with a Soft Gripper. Please check the device.<br>Program halted."
  sg_initialize_timeout="Gripper did not initialize in time!"

  #======    End of OnRobot SG Engine Messages Messages    ======#
  #======    OnRobot SG Engine    ======#

  sg_dataProcess_running=False
  def sg_dataProcess():
  enter_critical
  local tool_index=sg_index
  if tool_index==ON_DI_DUAL:
  sg_Width_primary=sg_Width_arr[ON_DI_PRIMARY]
  sg_Depth_primary=sg_Depth_arr[ON_DI_PRIMARY]
  sg_Busy_primary=sg_Busy_arr[ON_DI_PRIMARY]
  sg_Width_secondary=sg_Width_arr[ON_DI_SECONDARY]
  sg_Depth_secondary=sg_Depth_arr[ON_DI_SECONDARY]
  sg_Busy_secondary=sg_Busy_arr[ON_DI_SECONDARY]
  else:
  sg_Width=sg_Width_arr[tool_index]
  sg_Depth=sg_Depth_arr[tool_index]
  sg_Busy=sg_Busy_arr[tool_index]
  end
  exit_critical
  end
  def sg_dataProcess_status_errors(sg_stop=False):
  enter_critical
  local tool_index=sg_index
  if(tool_index==ON_DI_DUAL):
  tool_index=ON_DI_SECONDARY
  sg_stop=on_error((sg_device_id_arr[tool_index]!=tool_index),sg_status_error_missing,sg_status_error_title,sg_stop)
  sg_stop=on_error((sg_product_code_arr[tool_index]==ON_DEVICE_ID_MISSING),sg_status_error_missing,sg_status_error_title,sg_stop)
  tool_index=ON_DI_PRIMARY
  end
  sg_stop=on_error((sg_device_id_arr[tool_index]!=tool_index),sg_status_error_missing,sg_status_error_title,sg_stop)
  sg_stop=on_error((sg_product_code_arr[tool_index]==ON_DEVICE_ID_MISSING),sg_status_error_missing,sg_status_error_title,sg_stop)
  exit_critical
  return sg_stop
  end
  thread sg_dataProcess_thread():
  if ON_DEBUG_LOG:
  textmsg("Starting sg dataProcess thread")
  end
  while sg_dataProcess_running:
  sync()
  local sg_stop=False
  sg_stop=sg_dataProcess_status_errors(sg_stop)
  if sg_stop:
  halt
  end
  sg_dataProcess()
  end
  if ON_DEBUG_LOG:
  textmsg("Stopping sg dataProcess thread")
  end
  end

  #======    End of OnRobot SG Engine    ======#
  sg_tool_id_arr[0] = 1
  sg_Depth_arr[0] = 10.0
  textmsg(on_devices_primary_log, ": Quick Changer for I/O + SG + [0.0, 0.0, 0.0, 0.0, 0.0, 0.0]")
  on_follow_tcp = False
  on_tcp_active_is_primary = True
  on_tcp_adapters_array = []
  on_cog_adapters_array = []
  on_mass_adapters_array = []
  on_tcp_qc_primary = p[0.0, 0.0, 0.0196, 0.0, 0.0, 0.0]
  on_cog_qc_primary = p[0.0, 0.0, 0.007, 0.0, 0.0, 0.0]
  on_mass_qc_primary = 0.093
  on_tcp_gripper_static_primary = p[0.0, 0.0, 0.1339, 0.0, 0.0, 0.0]
  on_cog_gripper_primary = p[-0.012, -0.005, 0.050, 0.0, 0.0, 0.0]
  on_mass_gripper_primary = 1.01
  on_tcp_workpiece_primary = p[0.0, 0.0, 0.0, 0.0, 0.0, 0.0]
  on_cog_workpiece_primary = p[0.0, 0.0, 0.0, 0.0, 0.0, 0.0]
  on_mass_workpiece_primary = 0.0
  #======    OnRobot Soft Gripper Grip Messages    ======#

  sg_grip_error_title="OnRobot - Soft Gripper Grip error"
  sg_grip_title="OnRobot - Soft Gripper Grip"
  sg_grip_return_error="The Soft Gripper Grip command returned with error."
  sg_grip_return_0="The Grip command finished."

  #======    End of OnRobot Soft Gripper Grip Messages    ======#
  #======    OnRobot SG Grip    ======#

  def sg_wait_to_initialize(tool_index):
  local wait_timeout=ON_INIT_TIMEOUT
  while(wait_timeout>0):
  if sg_Initialized_arr[tool_index]:
  return 0
  else:
  sleep(0.008)
  wait_timeout=wait_timeout-1
  end
  end
  popup(sg_initialize_timeout,sg_error_title,error=True,blocking=False)
  halt
  end
  def sg_initialize(tool_index,sg_tool_id):
  on_tool_xmlrpc.sg_initialize(tool_index,sg_tool_id)
  sg_wait_to_initialize(tool_index)
  end
  def sg_depth_compensate(tool_index,start_depth_mm):
  local timeout=0
  while not sg_Busy_arr[tool_index]:
  sleep(0.008)
  timeout=timeout+1
  if timeout>20:
  break
  end
  end
  local start_pose=get_forward_kin()
  if(tool_index==ON_DI_SECONDARY):
  local tcp_static=on_tcp_static_secondary
  else:
  local tcp_static=on_tcp_static_primary
  end
  local t_w_rg=pose_trans(get_actual_tool_flange_pose(),tcp_static)
  local t_rg_w=pose_inv(t_w_rg)
  local compensation_depth_mm=0
  local after_ready_continue_count=10
  while True:
  local busy=sg_Busy_arr[tool_index]
  if not busy:
  if after_ready_continue_count>0:
  after_ready_continue_count=after_ready_continue_count-1
  else:
  break
  end
  end
  local measure_depth_mm=sg_Depth_arr[tool_index]
  compensation_depth_mm=measure_depth_mm-start_depth_mm
  local target_pose=pose_add(start_pose,pose_trans(pose_trans(t_w_rg,p[0,0,compensation_depth_mm/1000.0,0,0,0]),t_rg_w))
  servoj(get_inverse_kin(target_pose),t=0.008,lookahead_time=0.033,gain=1500)
  end
  stopj(20)
  end
  def sg_wait_for_move(tool_index):
  local timeout=0
  while not sg_Busy_arr[tool_index]:
  sleep(0.008)
  timeout=timeout+1
  if timeout>20:
  break
  end
  end
  local after_ready_continue_count=10
  while True:
  local busy=sg_Busy_arr[tool_index]
  if not busy:
  if after_ready_continue_count>0:
  after_ready_continue_count=after_ready_continue_count-1
  else:
  break
  end
  end
  end
  end
  def sg_grip(target_width,gentle_grip,tool_index=0,blocking=True,depth_compensation=False):
  sg_Grip_command_arr[tool_index]=True
  return sg_width(target_width,gentle_grip,tool_index,blocking,depth_compensation,True)
  end
  def sg_release(target_width,tool_index=0,blocking=True,depth_compensation=False):
  sg_Grip_command_arr[tool_index]=False
  return sg_width(target_width,False,tool_index,blocking,depth_compensation,False)
  end
  def sg_width(target_width,gentle_grip,tool_index=0,blocking=True,depth_compensation=False,is_grip=False):
  if ON_DEBUG_LOG:
  textmsg("SG Grip start..")
  end
  local retVal=0
  if not sg_Initialized_arr[tool_index]:
  sg_initialize(tool_index,sg_tool_id_arr[tool_index])
  end
  if depth_compensation:
  local start_depth_mm=sg_Depth_arr[tool_index]
  end
  retVal=on_tool_xmlrpc.sg_grip(tool_index,target_width,gentle_grip,is_grip)
  if(retVal!=0):
  popup(sg_grip_return_error,sg_grip_error_title,error=True,blocking=False)
  halt
  end
  if blocking:
  if depth_compensation:
  sg_depth_compensate(tool_index,start_depth_mm)
  else:
  sg_wait_for_move(tool_index)
  end
  end
  sync()
  return retVal
  end

  #======    End of OnRobot SG Grip    ======#
  #======    OnRobot WebLytics Messages    ======#

  wl_weblytics_message_title="OnRobot - Weblytics"
  wl_start_stop_section_error_command="Could not send set variable command<br>Please check connection.<br>Program halted."

  #======    End of OnRobot WebLytics Messages    ======#
  #======    OnRobot WebLytics    ======#

  def wl_increment_variable(register):
  on_conn_xmlrpc.cb_increment_weblytics_variable(register,1)
  end
  def wl_start_stop_section(section):
  local err=on_conn_xmlrpc.cb_set_weblytics_variable(32768,section)
  if err<0:
  popup(wl_start_stop_section_error_command,title=wl_weblytics_message_title,error=True,blocking=False)
  halt
  end
  end

  #======    End of OnRobot WebLytics    ======#
  #======    OnRobot Run    ======#

  on_portopen_javaSocket()
  sync()
  textmsg(on_xmlrpc_start_ip,on_conn_ip)
  if(ON_REG_USE_TOOL):
  on_regStart_conn=[ON_CONN_SHIFT_BOOL,ON_CONN_SHIFT_INT,ON_CONN_SHIFT_FLOAT]
  on_regSum_conn=[ON_CONN_REG_SUM_BOOL,ON_CONN_REG_SUM_INT,ON_CONN_REG_SUM_FLOAT]
  on_rtde_feed_open(on_conn_ip,on_conn_rtde_feed_name,on_regStart_conn,on_regSum_conn,ON_REGISTERS_SPEEDL_FLOAT)
  sync()
  textmsg(on_xmlrpc_start_ip,on_tool_ip)
  on_regStart_tool=[ON_TOOL_SHIFT_BOOL,ON_TOOL_SHIFT_INT,ON_TOOL_SHIFT_FLOAT]
  on_regSum_tool=[ON_TOOL_REG_SUM_BOOL,ON_TOOL_REG_SUM_INT,ON_TOOL_REG_SUM_FLOAT]
  on_rtde_feed_open(on_tool_ip,on_tool_rtde_feed_name,on_regStart_tool,on_regSum_tool,0)
  sync()
  else:
  on_regStart_conn=[ON_CONN_SHIFT_BOOL,ON_CONN_SHIFT_INT,ON_CONN_SHIFT_FLOAT]
  on_regSum_conn=[ON_CONN_REG_SUM_BOOL,ON_CONN_REG_SUM_INT,ON_CONN_REG_SUM_FLOAT]
  on_rtde_feed_open(on_conn_ip,on_conn_rtde_feed_name,on_regStart_conn,on_regSum_conn,ON_REGISTERS_SPEEDL_FLOAT)
  sync()
  end
  on_set_rtde_watchdog(updateHz=0.2)
  sync()
  on_dataProcess_thrd=run on_dataProcess_thread()
  sync()
  on_tcp_init_adapters()
  on_payload_init_adapters()
  on_tcp_init_primary()
  on_payload_init_primary()

  on_tcp_update_custom()
  on_tcp_set_actual_to(on_tcp_active_is_primary)
  if(on_follow_tcp):
  on_payload_set_actual()
  end
  on_watchdog_thrd=run on_set_watchdog_thread()
  sync()
  def done_waiting_for_init(device_name,product_code,tool_index=0):
  textmsg(str_cat(device_name,str_cat(str_cat("[",tool_index),"]: ")),product_code)
  end

  #======    End of OnRobot Run    ======#
  #======    OnRobot QC Start    ======#

  if(on_toolConnector):
  tc_setup_tool()
  end
  sync()

  #======    End of OnRobot QC Start    ======#
  #======    OnRobot SG Run    ======#

  def sg_wait_for_init(tool_index):
  local sg_timeout=0
  while not(sg_product_code_arr[tool_index]==SG_DEVICE_ID):
  sync()
  sg_timeout=sg_timeout+1
  if(sg_timeout>ON_INIT_TIMEOUT):
  popup(sg_status_error_missing,sg_status_error_title,error=True,blocking=False)
  halt
  end
  end
  done_waiting_for_init("SG",sg_product_code_arr[tool_index],tool_index)
  end
  sg_dataProcess_running=True
  sg_dataRead_running=True
  sync()
  sg_dataRead_thrd=run sg_dataRead_thread()
  sync()
  if(sg_index==ON_DI_DUAL):
  sg_wait_for_init(ON_DI_PRIMARY)
  sg_wait_for_init(ON_DI_SECONDARY)
  else:
  sg_wait_for_init(sg_index)
  end
  sync()
  sg_dataProcess_thrd=run sg_dataProcess_thread()
  sync()

  #======    End of OnRobot SG Run    ======#
  #======    OnRobot WL Run    ======#

  if on_computebox:
  on_conn_xmlrpc.cb_set_weblytics_variables(32768,32870,0)
  end

  #======    End of OnRobot WL Run    ======#
  # end: URCap Installation Node
  $ 1 "BeforeStart"
  $ 2 "MoveJ"
  $ 3 "Waypoint_1" "breakAfter"
  movej(get_inverse_kin(p[-.159567213765, -.023556580058, .496075585500, .029228760514, .015566801012, .875879801508], qnear=[-0.6221788565265101, -0.1537726561175745, -2.6713267008410853, 1.2235838174819946, 1.5651061534881592, 3.069310188293457]), a=1.3962634015954636, v=1.0471975511965976)
  # begin: URCap Program Node
  #   Source: OnRobot, 6.0.3, OnRobot A/S
  #   Type: SG Grip
  $ 4 "SG Grip (86)"
on_return = sg_grip(86, True, tool_index = 0, blocking = True, depth_compensation = False)
sg_payload_set(mass = 0.0, tool_index = 0)
  # end: URCap Program Node
  while (True):
    $ 5 "Robot Program"
    $ 6 "var_1≔'vino rosso:1, vino bianco:2'"
    global var_1=request_integer_from_primary_client("vino rosso:1, vino bianco:2")
    $ 7 "If var_1==1"
    if (var_1==1):
      $ 8 "MoveJ"
      $ 9 "appr" "breakAfter"
      movej(get_inverse_kin(p[.025586625574, -.217556890987, .345360944179, 2.196698062048, 1.496905624061, -.006385815850], qnear=[-0.8226197401629847, -0.9496062437640589, -1.300997559224264, -1.982403580342428, 1.4991928339004517, 2.6763968467712402]), a=1.3962634015954636, v=1.0471975511965976)
      $ 10 "Waypoint_2" "breakAfter"
      movej(get_inverse_kin(p[.031418776545, -.217434087568, .324643713019, 2.245998536330, 1.499443680924, .017514345782], qnear=[-0.8228710333453577, -0.937843147908346, -1.3946316877948206, -1.9407208601581019, 1.5178706645965576, 2.70094633102417]), a=1.3962634015954636, v=1.0471975511965976)
      # begin: URCap Program Node
      #   Source: OnRobot, 6.0.3, OnRobot A/S
      #   Type: SG Grip
      $ 11 "SG Grip (20)"
on_return = sg_grip(20, True, tool_index = 0, blocking = True, depth_compensation = False)
sg_payload_set(mass = 2.0, tool_index = 0)
      # end: URCap Program Node
      $ 12 "Waypoint_3" "breakAfter"
      movej(get_inverse_kin(p[.031205663451, -.218665145534, .347337893823, 2.291334910493, 1.532821010629, -.000149611036], qnear=[-0.8229430357562464, -1.0759480635272425, -1.1508773008929651, -2.103816811238424, 1.5136147737503052, 2.699615001678467]), a=1.3962634015954636, v=1.0471975511965976)
      $ 13 "Waypoint_4" "breakAfter"
      movej(get_inverse_kin(p[-.044404960955, -.119171549305, .429402905550, 1.904681866833, 1.293164257612, .145598424445], qnear=[-0.8234341780291956, -0.7063797155963343, -0.905313793812887, -2.255631748829977, 1.5653338432312012, 2.693235158920288]), a=1.3962634015954636, v=1.0471975511965976)
      $ 14 "MoveJ"
      $ 15 "Waypoint_5" "breakAfter"
      movej(get_inverse_kin(p[.020049672808, .142744402797, .658935309121, 1.245353604590, -1.633965634543, -1.981834782440], qnear=[-3.80415922800173, -1.2332118193255823, 0.07471990585327148, -1.996488396321432, 1.5185058116912842, 2.695093870162964]), a=1.3962634015954636, v=1.0471975511965976)
      $ 16 "Wait: 2.0"
      sleep(2.0)
      $ 17 "Waypoint_6" "breakAfter"
      movej(get_inverse_kin(p[.009998353263, .150467735493, .547731276946, 1.543656684275, -1.985793853107, -1.527407719536], qnear=[-3.804099146519796, -1.2348769346820276, 0.07449197769165039, -2.4436100164996546, 1.5184818506240845, 2.695573091506958]), a=1.3962634015954636, v=1.0471975511965976)
      $ 18 "Wait: 1.0"
      sleep(1.0)
      $ 19 "Waypoint_7" "breakAfter"
      movej(get_inverse_kin(p[.020074859306, .142735506047, .658922595777, 1.245405381310, -1.633990935906, -1.981880845629], qnear=[-3.80415922800173, -1.2331398169146937, 0.07469558715820312, -1.9965480009662073, 1.5184699296951294, 2.6950340270996094]), a=1.3962634015954636, v=1.0471975511965976)
      $ 20 "MoveJ"
      $ 21 "Waypoint_8" "breakAfter"
      movej(get_inverse_kin(p[-.043492485474, -.137421776727, .658955234025, 1.339416104693, .854336962482, .190144844203], qnear=[-0.8295076529132288, -1.2332237402545374, 0.07474374771118164, -1.9964163939105433, 1.5185178518295288, 2.695081949234009]), a=1.3962634015954636, v=1.0471975511965976)
      $ 22 "Waypoint_9" "breakAfter"
      movej(get_inverse_kin(p[-.046795952823, -.133622679054, .408730488837, 1.922741619412, 1.265150078414, .092816107569], qnear=[-0.8228352705584925, -0.6132867972003382, -1.1087830702411097, -2.148716751729147, 1.5164557695388794, 2.7008862495422363]), a=1.3962634015954636, v=1.0471975511965976)
      $ 23 "Waypoint_10" "breakAfter"
      movej(get_inverse_kin(p[.031440500239, -.217419557689, .324617822402, 2.245974257556, 1.499639011592, .017566258598], qnear=[-0.8227751890765589, -0.9378312269793909, -1.3947036902057093, -1.940744702016012, 1.517906665802002, 2.7009222507476807]), a=1.3962634015954636, v=1.0471975511965976)
      # begin: URCap Program Node
      #   Source: OnRobot, 6.0.3, OnRobot A/S
      #   Type: SG Release
      $ 24 "SG Release (80)"
on_return = sg_release(80, tool_index = 0, blocking = True, depth_compensation = False)
sg_payload_set(mass = 0.0, tool_index = 0)
      # end: URCap Program Node
    else:
      $ 25 "ElseIf var_1==2"
      if (var_1==2):
        $ 26 "MoveJ"
        $ 27 "Waypoint_11" "breakAfter"
        movej(get_inverse_kin(p[.161964441376, -.156645543656, .337879999342, 1.271683833490, 2.605180516739, -.069970256395], qnear=[-0.0807722250567835, -1.2082393805133265, -1.0078538099872034, -2.2861889044391077, 1.440742015838623, 2.384781837463379]), a=1.3962634015954636, v=1.0471975511965976)
        $ 28 "Waypoint_12" "breakAfter"
        movej(get_inverse_kin(p[.163817257934, -.158290958428, .322528630889, 1.222504808441, 2.715047887419, -.134121680130], qnear=[-0.08073646226991826, -1.2527230421649378, -1.0272701422320765, -2.308791462575094, 1.4344252347946167, 2.328078508377075]), a=1.3962634015954636, v=1.0471975511965976)
        # begin: URCap Program Node
        #   Source: OnRobot, 6.0.3, OnRobot A/S
        #   Type: SG Grip
        $ 29 "SG Grip (20)"
on_return = sg_grip(20, True, tool_index = 0, blocking = True, depth_compensation = False)
sg_payload_set(mass = 2.0, tool_index = 0)
        # end: URCap Program Node
        $ 30 "Waypoint_14" "breakAfter"
        movej(get_inverse_kin(p[.162610355263, -.154735168406, .362751151258, 1.187272569445, 2.632213436879, -.059572766173], qnear=[-0.08139545122255498, -1.3004158178912562, -0.7787888685809534, -2.4058082739459437, 1.4494324922561646, 2.323127508163452]), a=1.3962634015954636, v=1.0471975511965976)
        $ 31 "Waypoint_15" "breakAfter"
        movej(get_inverse_kin(p[.102370640034, -.145268413102, .478205162862, .933348742503, 2.196656670968, .163669877782], qnear=[-0.0814436117755335, -1.205376927052633, -0.2573445479022425, -2.4926980177508753, 1.4687799215316772, 2.2521040439605713]), a=1.3962634015954636, v=1.0471975511965976)
        $ 32 "Waypoint_16" "breakAfter"
        movej(get_inverse_kin(p[.020042058691, .142768651175, .658926198216, 1.245351259585, -1.634056890254, -1.981789660845], qnear=[-3.8041232267962855, -1.2332356611834925, 0.0747079849243164, -1.9965117613421839, 1.518433928489685, 2.695117712020874]), a=1.3962634015954636, v=1.0471975511965976)
      end
    end
  end
end
